// TIA Portal V19 export
VAR_GLOBAL   // PLC tag table "U2Em5_Output"
   trayLiftingCylinderWorkPositionU2Em5 AT %Q46.0 : Bool;   // U2Em5_ Plastic tray lifting cylinder working position / Em120_塑胶托盘顶升气缸工作位
   trayLiftingCylinderHomePositionU2Em5 AT %Q46.1 : Bool;   // U2Em5_ Plastic tray lifting cylinder in situ / Em120_塑胶托盘顶升气缸原位
END_VAR
